(* Logix 5000 project; controller Sucrose_Main Emulate 5570 rev 20.12; software revision 20.01; part 11 of 30 *)
(* tags used below, declared in another part *)
   AI_E21_1 : REAL[8];   // Analog Input EN2T_FLX 192.168.1.21
   AI_E21_2 : REAL[8];   // Analog Input EN2T_FLX 192.168.1.21
   AI_E23_1 : REAL[8];   // Analog Input EN2T_FLX 192.168.1.23
   Alarm_ACK_Master_Timer : TIMER;
   ClearFault_Master : BOOL;
   DI_E20_2 : ALIAS FOR FLX_E20:2:I;   // Discrete Input EN2T_FLX 192.168.1.20
   DO_E24_3 : ALIAS FOR FLX_E24:3:O;   // Discrete Output EN2T_FLX 192.168.1.24
   FV230303_AOI : QSI_Flow_Valve;   // FV-23-03-03 SUCROSE TANK #3 OUTLET VALVE
   HEADER_FLOW_SP : DINT;
   ONESHOTBITS : INT[10];
   P230401_AOI : PF525_VFD_E_ENET;   // P-23-04-01 SUCROSE TRANSFER PUMP 1
   P230402_AOI : PF525_VFD_E_ENET;   // P-23-04-02 SUCROSE TRANSFER PUMP 2
   READ_FROM_SUCROSE_CIP : DINT[10];
   Rung_Comment : BOOL;
   Sucrose_MM_Enable : BOOL;
   SucroseCIP_FILTRATION_REMOTE : CIP_REMOTE;
   SucroseCIP_P230401_REMOTE : CIP_REMOTE;
   SucroseCIP_P230402_REMOTE : CIP_REMOTE;
   SucroseCIP_TK230301_REMOTE : CIP_REMOTE;
   SucroseDischarge : Area_Program;
   SucroseFiltration : Area_Program;
   SucroseTanks : Area_Program;
   temp_toggle : BOOL;
   toggle : BOOL;
(* DischargeArea_EN2T_IO_Discrete_DO_E24_3, continued *)

ROUTINE _11_FV230303   (* ladder *)
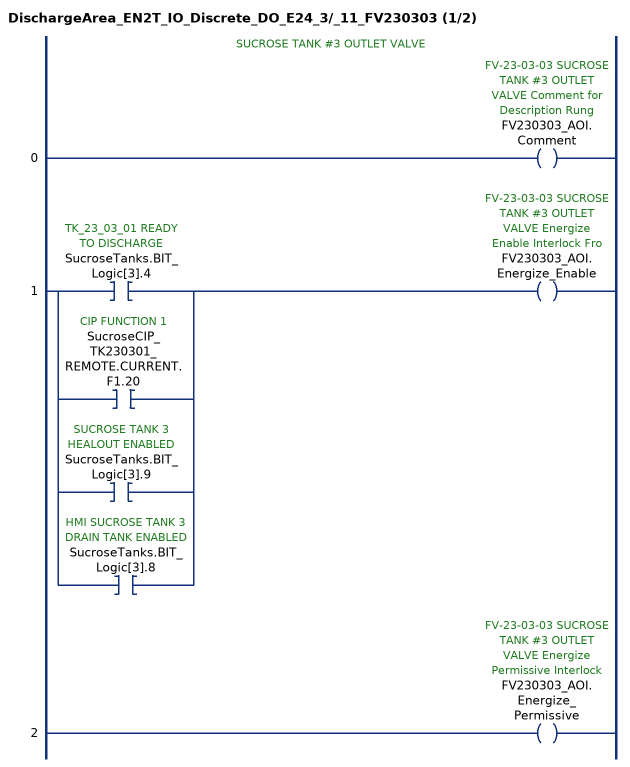
   // SUCROSE TANK #3 OUTLET VALVE
   0: OTE(FV230303_AOI.Comment);
   1: [XIC(SucroseTanks.BIT_Logic[3].4) ,XIC(SucroseCIP_TK230301_REMOTE.CURRENT.F1.20) ,XIC(SucroseTanks.BIT_Logic[3].9) ,XIC(SucroseTanks.BIT_Logic[3].8) ]OTE(FV230303_AOI.Energize_Enable);
   2: OTE(FV230303_AOI.Energize_Permissive);
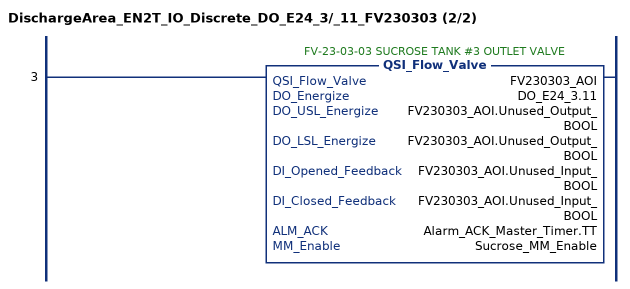
   3: QSI_Flow_Valve(FV230303_AOI,DO_E24_3.11,FV230303_AOI.Unused_Output_BOOL,FV230303_AOI.Unused_Output_BOOL,FV230303_AOI.Unused_Input_BOOL,FV230303_AOI.Unused_Input_BOOL,Alarm_ACK_Master_Timer.TT,Sucrose_MM_Enable);
END_ROUTINE

ROUTINE MainRoutine   (* ladder *)
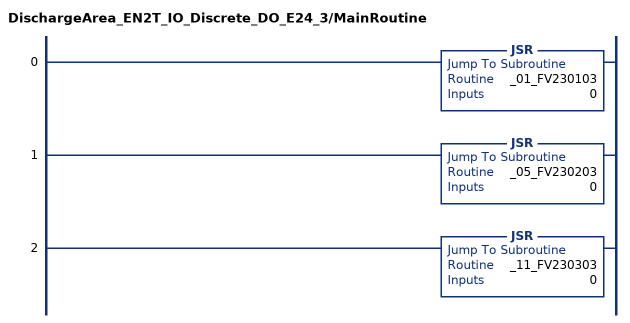
   0: JSR(_01_FV230103,0);
   1: JSR(_05_FV230203,0);
   2: JSR(_11_FV230303,0);
END_ROUTINE
END_PROGRAM

PROGRAM DischargeArea_EN2T_IO_Drives   (* main routine MainRoutine *)

ROUTINE E30_P230401   (* ladder *)
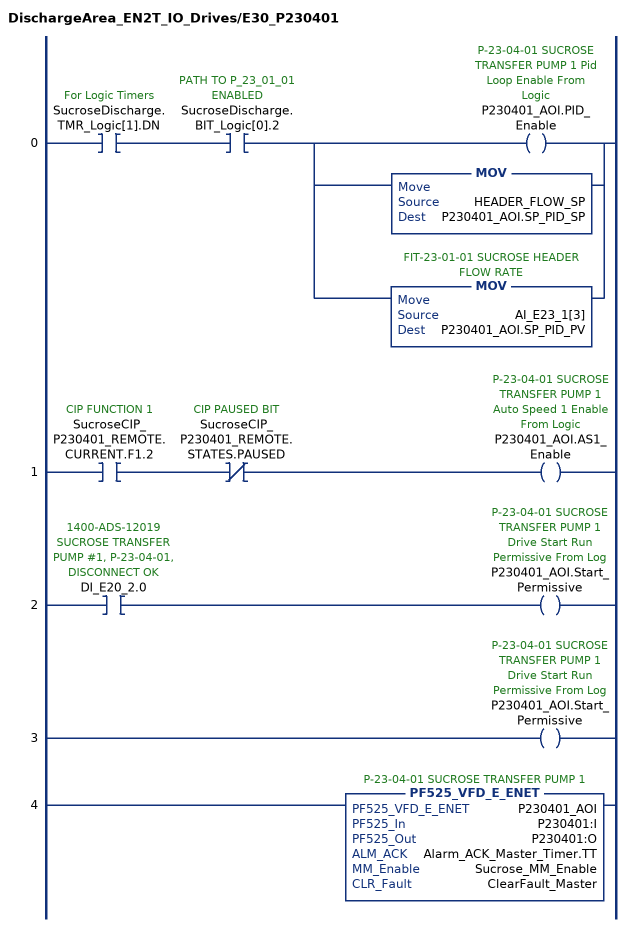
   0: XIC(SucroseDischarge.TMR_Logic[1].DN)XIC(SucroseDischarge.BIT_Logic[0].2)[OTE(P230401_AOI.PID_Enable) ,MOV(HEADER_FLOW_SP,P230401_AOI.SP_PID_SP) ,MOV(AI_E23_1[3],P230401_AOI.SP_PID_PV) ];
   1: XIC(SucroseCIP_P230401_REMOTE.CURRENT.F1.2)XIO(SucroseCIP_P230401_REMOTE.STATES.PAUSED)OTE(P230401_AOI.AS1_Enable);
   2: XIC(DI_E20_2.0)OTE(P230401_AOI.Start_Permissive);
   3: OTE(P230401_AOI.Start_Permissive);
   4: PF525_VFD_E_ENET(P230401_AOI,P230401:I,P230401:O,Alarm_ACK_Master_Timer.TT,Sucrose_MM_Enable,ClearFault_Master);
END_ROUTINE

ROUTINE E31_P200402   (* ladder *)
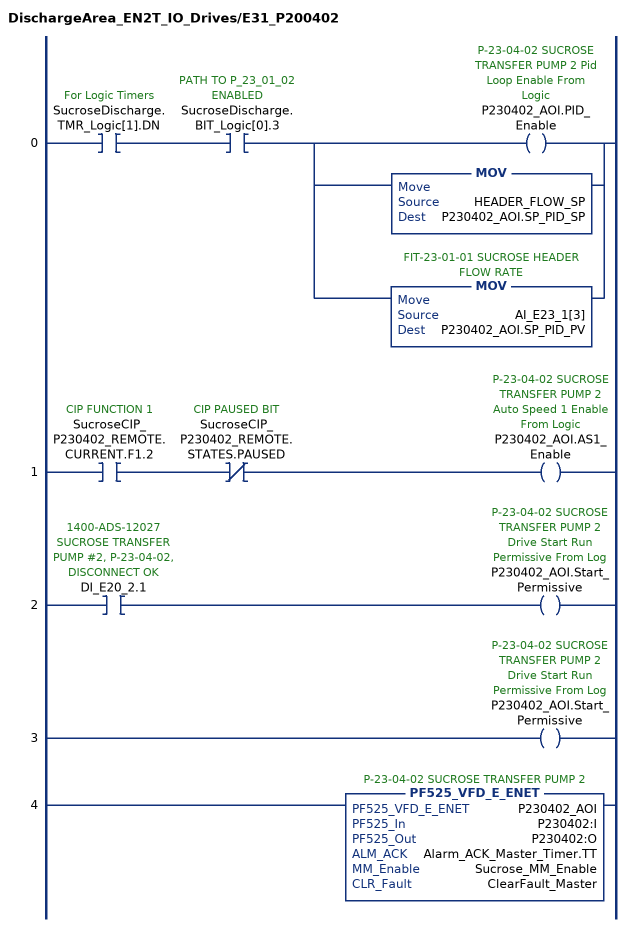
   0: XIC(SucroseDischarge.TMR_Logic[1].DN)XIC(SucroseDischarge.BIT_Logic[0].3)[OTE(P230402_AOI.PID_Enable) ,MOV(HEADER_FLOW_SP,P230402_AOI.SP_PID_SP) ,MOV(AI_E23_1[3],P230402_AOI.SP_PID_PV) ];
   1: XIC(SucroseCIP_P230402_REMOTE.CURRENT.F1.2)XIO(SucroseCIP_P230402_REMOTE.STATES.PAUSED)OTE(P230402_AOI.AS1_Enable);
   2: XIC(DI_E20_2.1)OTE(P230402_AOI.Start_Permissive);
   3: OTE(P230402_AOI.Start_Permissive);
   4: PF525_VFD_E_ENET(P230402_AOI,P230402:I,P230402:O,Alarm_ACK_Master_Timer.TT,Sucrose_MM_Enable,ClearFault_Master);
END_ROUTINE

ROUTINE MainRoutine   (* ladder *)
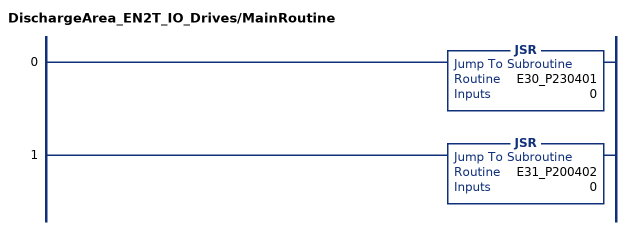
   0: JSR(E30_P230401,0);
   1: JSR(E31_P200402,0);
END_ROUTINE
END_PROGRAM

PROGRAM FiltrationArea_AutoLogic   (* main routine MainRoutine *)

ROUTINE Alarm_Logic   (* ladder *)
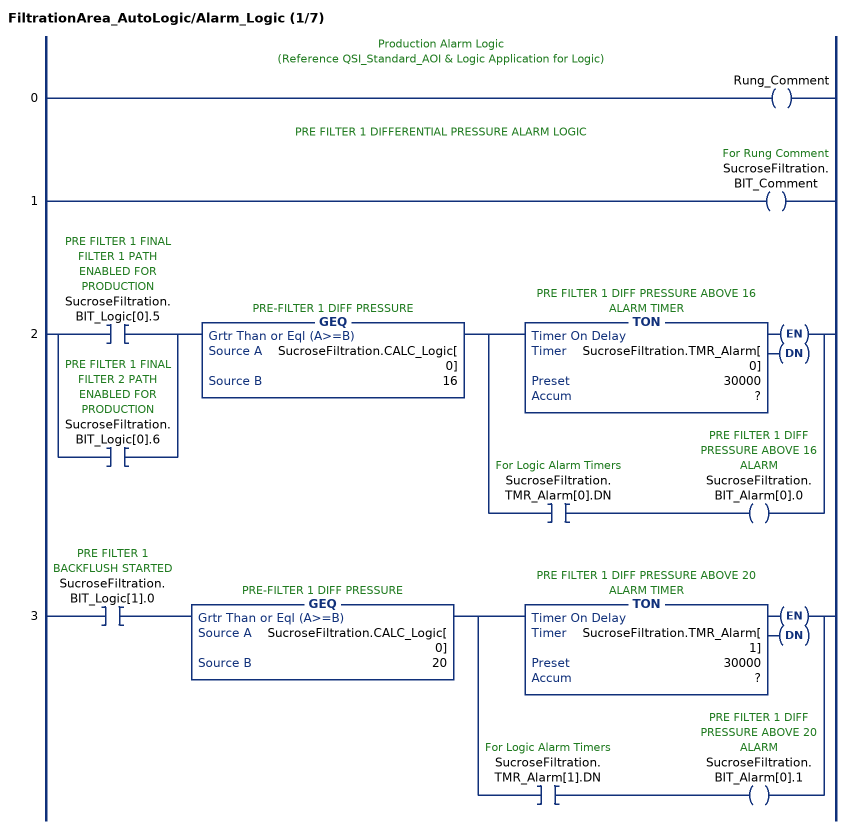
   // Production Alarm Logic
   // (Reference QSI_Standard_AOI & Logic Application for Logic)
   0: OTE(Rung_Comment);
   // PRE FILTER 1 DIFFERENTIAL PRESSURE ALARM LOGIC
   1: OTE(SucroseFiltration.BIT_Comment);
   2: [XIC(SucroseFiltration.BIT_Logic[0].5) ,XIC(SucroseFiltration.BIT_Logic[0].6) ]GEQ(SucroseFiltration.CALC_Logic[0],16)[TON(SucroseFiltration.TMR_Alarm[0],?,?) ,XIC(SucroseFiltration.TMR_Alarm[0].DN) OTE(SucroseFiltration.BIT_Alarm[0].0) ];
   3: XIC(SucroseFiltration.BIT_Logic[1].0)GEQ(SucroseFiltration.CALC_Logic[0],20)[TON(SucroseFiltration.TMR_Alarm[1],?,?) ,XIC(SucroseFiltration.TMR_Alarm[1].DN) OTE(SucroseFiltration.BIT_Alarm[0].1) ];
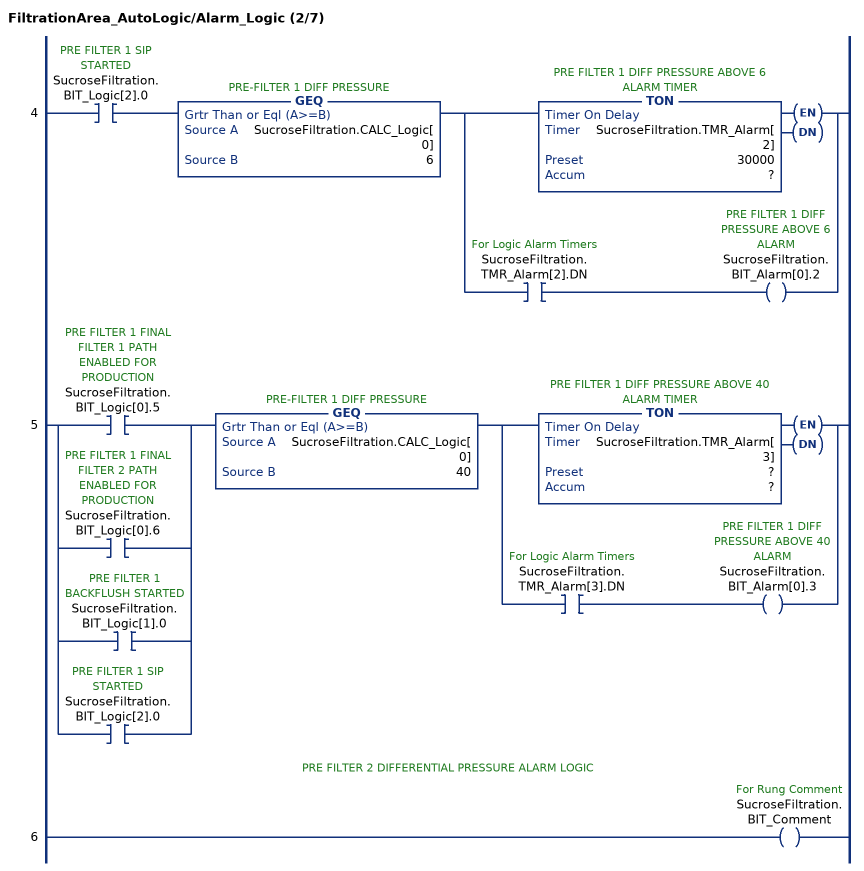
   4: XIC(SucroseFiltration.BIT_Logic[2].0)GEQ(SucroseFiltration.CALC_Logic[0],6)[TON(SucroseFiltration.TMR_Alarm[2],?,?) ,XIC(SucroseFiltration.TMR_Alarm[2].DN) OTE(SucroseFiltration.BIT_Alarm[0].2) ];
   5: [XIC(SucroseFiltration.BIT_Logic[0].5) ,XIC(SucroseFiltration.BIT_Logic[0].6) ,XIC(SucroseFiltration.BIT_Logic[1].0) ,XIC(SucroseFiltration.BIT_Logic[2].0) ]GEQ(SucroseFiltration.CALC_Logic[0],40)[TON(SucroseFiltration.TMR_Alarm[3],?,?) ,XIC(SucroseFiltration.TMR_Alarm[3].DN) OTE(SucroseFiltration.BIT_Alarm[0].3) ];
   // PRE FILTER 2 DIFFERENTIAL PRESSURE ALARM LOGIC
   6: OTE(SucroseFiltration.BIT_Comment);
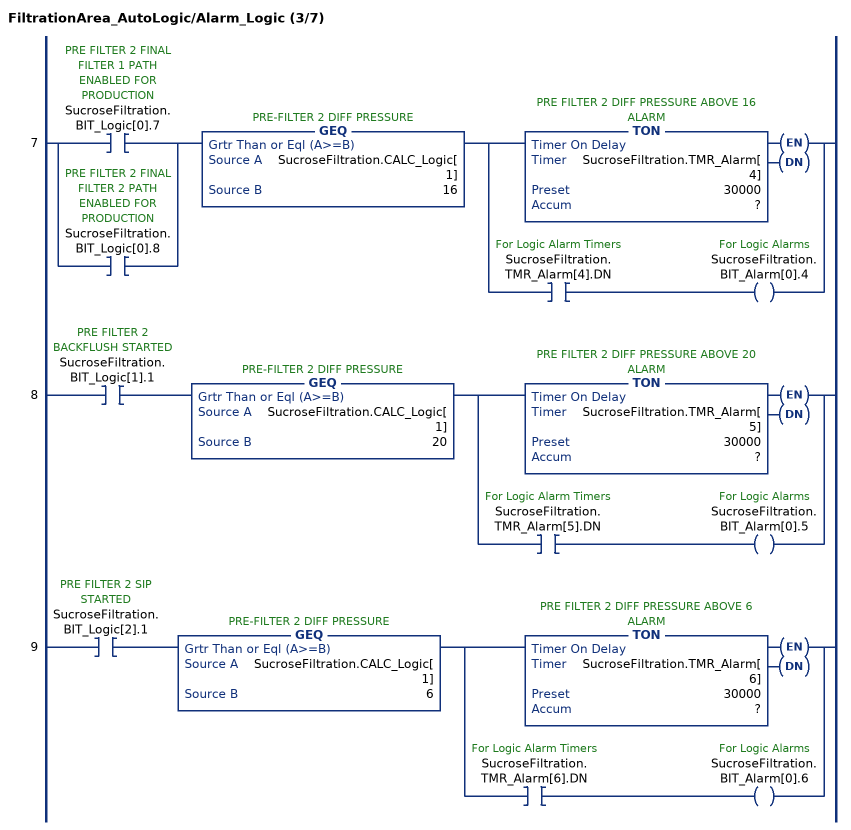
   7: [XIC(SucroseFiltration.BIT_Logic[0].7) ,XIC(SucroseFiltration.BIT_Logic[0].8) ]GEQ(SucroseFiltration.CALC_Logic[1],16)[TON(SucroseFiltration.TMR_Alarm[4],?,?) ,XIC(SucroseFiltration.TMR_Alarm[4].DN) OTE(SucroseFiltration.BIT_Alarm[0].4) ];
   8: XIC(SucroseFiltration.BIT_Logic[1].1)GEQ(SucroseFiltration.CALC_Logic[1],20)[TON(SucroseFiltration.TMR_Alarm[5],?,?) ,XIC(SucroseFiltration.TMR_Alarm[5].DN) OTE(SucroseFiltration.BIT_Alarm[0].5) ];
   9: XIC(SucroseFiltration.BIT_Logic[2].1)GEQ(SucroseFiltration.CALC_Logic[1],6)[TON(SucroseFiltration.TMR_Alarm[6],?,?) ,XIC(SucroseFiltration.TMR_Alarm[6].DN) OTE(SucroseFiltration.BIT_Alarm[0].6) ];
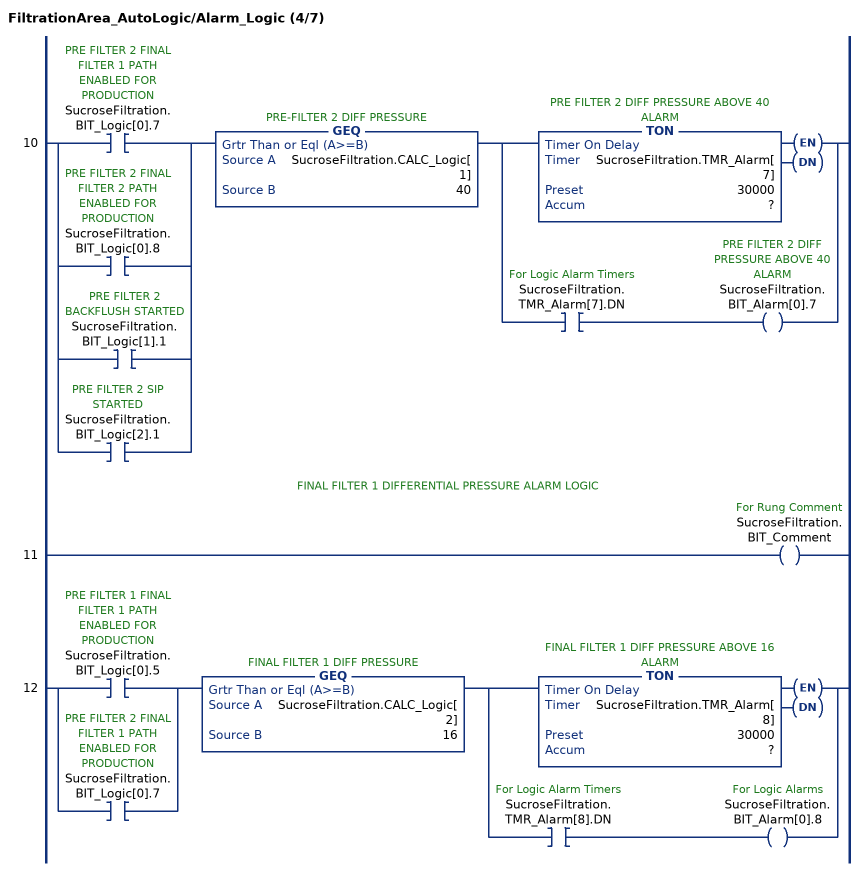
   10: [XIC(SucroseFiltration.BIT_Logic[0].7) ,XIC(SucroseFiltration.BIT_Logic[0].8) ,XIC(SucroseFiltration.BIT_Logic[1].1) ,XIC(SucroseFiltration.BIT_Logic[2].1) ]GEQ(SucroseFiltration.CALC_Logic[1],40)[TON(SucroseFiltration.TMR_Alarm[7],?,?) ,XIC(SucroseFiltration.TMR_Alarm[7].DN) OTE(SucroseFiltration.BIT_Alarm[0].7) ];
   // FINAL FILTER 1 DIFFERENTIAL PRESSURE ALARM LOGIC
   11: OTE(SucroseFiltration.BIT_Comment);
   12: [XIC(SucroseFiltration.BIT_Logic[0].5) ,XIC(SucroseFiltration.BIT_Logic[0].7) ]GEQ(SucroseFiltration.CALC_Logic[2],16)[TON(SucroseFiltration.TMR_Alarm[8],?,?) ,XIC(SucroseFiltration.TMR_Alarm[8].DN) OTE(SucroseFiltration.BIT_Alarm[0].8) ];
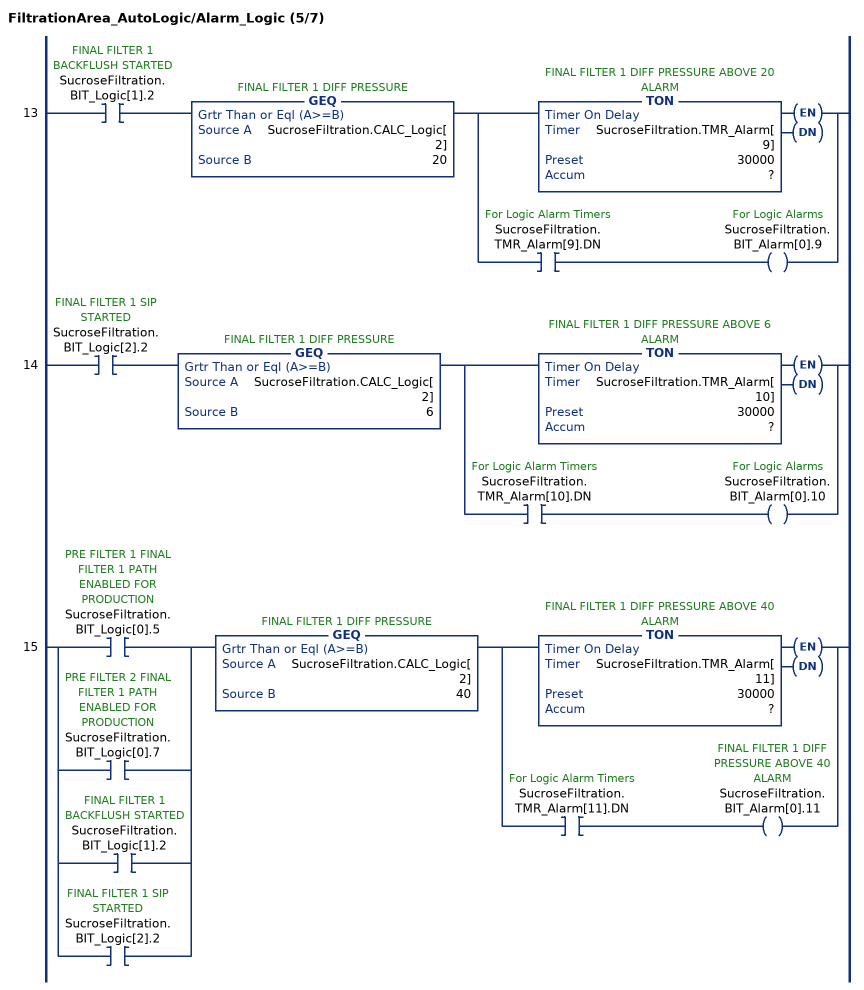
   13: XIC(SucroseFiltration.BIT_Logic[1].2)GEQ(SucroseFiltration.CALC_Logic[2],20)[TON(SucroseFiltration.TMR_Alarm[9],?,?) ,XIC(SucroseFiltration.TMR_Alarm[9].DN) OTE(SucroseFiltration.BIT_Alarm[0].9) ];
   14: XIC(SucroseFiltration.BIT_Logic[2].2)GEQ(SucroseFiltration.CALC_Logic[2],6)[TON(SucroseFiltration.TMR_Alarm[10],?,?) ,XIC(SucroseFiltration.TMR_Alarm[10].DN) OTE(SucroseFiltration.BIT_Alarm[0].10) ];
   15: [XIC(SucroseFiltration.BIT_Logic[0].5) ,XIC(SucroseFiltration.BIT_Logic[0].7) ,XIC(SucroseFiltration.BIT_Logic[1].2) ,XIC(SucroseFiltration.BIT_Logic[2].2) ]GEQ(SucroseFiltration.CALC_Logic[2],40)[TON(SucroseFiltration.TMR_Alarm[11],?,?) ,XIC(SucroseFiltration.TMR_Alarm[11].DN) OTE(SucroseFiltration.BIT_Alarm[0].11) ];
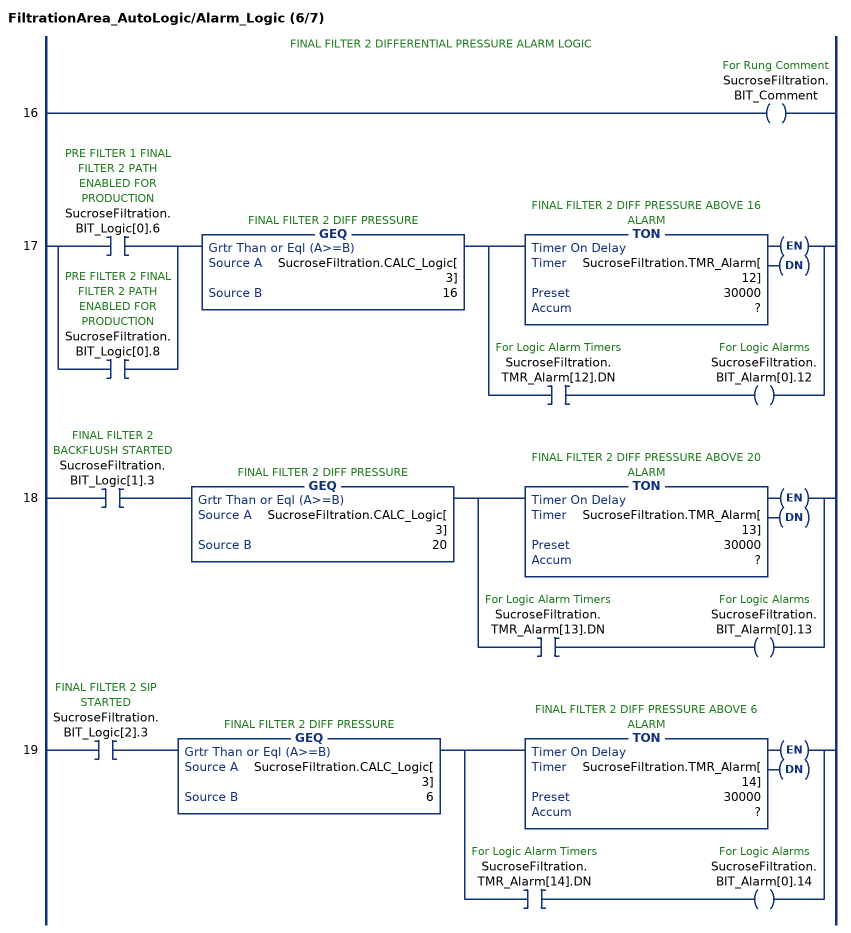
   // FINAL FILTER 2 DIFFERENTIAL PRESSURE ALARM LOGIC
   16: OTE(SucroseFiltration.BIT_Comment);
   17: [XIC(SucroseFiltration.BIT_Logic[0].6) ,XIC(SucroseFiltration.BIT_Logic[0].8) ]GEQ(SucroseFiltration.CALC_Logic[3],16)[TON(SucroseFiltration.TMR_Alarm[12],?,?) ,XIC(SucroseFiltration.TMR_Alarm[12].DN) OTE(SucroseFiltration.BIT_Alarm[0].12) ];
   18: XIC(SucroseFiltration.BIT_Logic[1].3)GEQ(SucroseFiltration.CALC_Logic[3],20)[TON(SucroseFiltration.TMR_Alarm[13],?,?) ,XIC(SucroseFiltration.TMR_Alarm[13].DN) OTE(SucroseFiltration.BIT_Alarm[0].13) ];
   19: XIC(SucroseFiltration.BIT_Logic[2].3)GEQ(SucroseFiltration.CALC_Logic[3],6)[TON(SucroseFiltration.TMR_Alarm[14],?,?) ,XIC(SucroseFiltration.TMR_Alarm[14].DN) OTE(SucroseFiltration.BIT_Alarm[0].14) ];
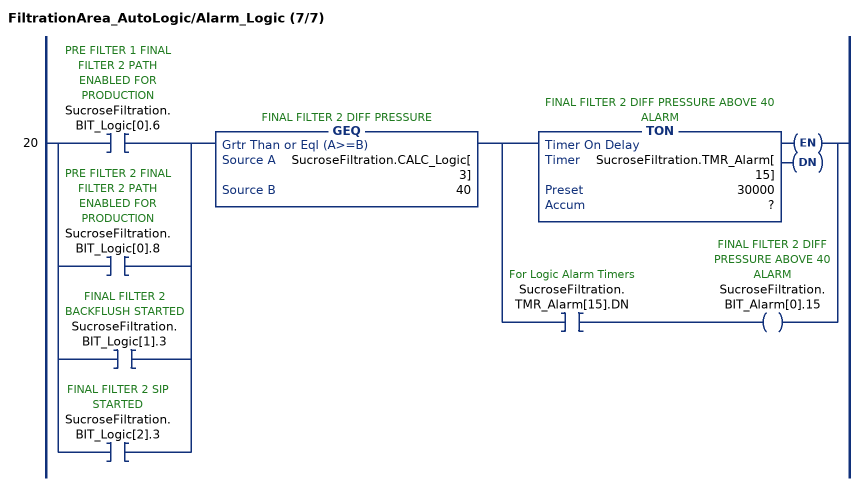
   20: [XIC(SucroseFiltration.BIT_Logic[0].6) ,XIC(SucroseFiltration.BIT_Logic[0].8) ,XIC(SucroseFiltration.BIT_Logic[1].3) ,XIC(SucroseFiltration.BIT_Logic[2].3) ]GEQ(SucroseFiltration.CALC_Logic[3],40)[TON(SucroseFiltration.TMR_Alarm[15],?,?) ,XIC(SucroseFiltration.TMR_Alarm[15].DN) OTE(SucroseFiltration.BIT_Alarm[0].15) ];
END_ROUTINE

ROUTINE Control_Logic   (* ladder *)
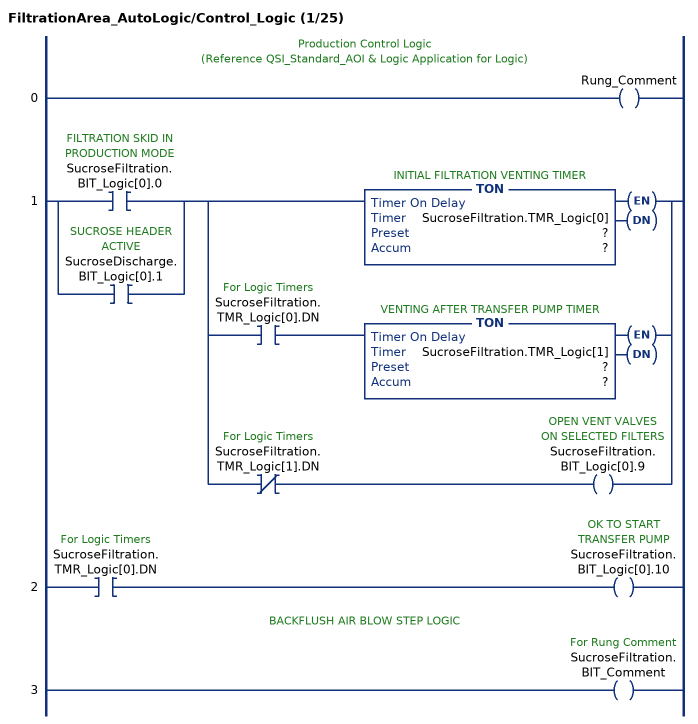
   // Production Control Logic
   // (Reference QSI_Standard_AOI & Logic Application for Logic)
   0: OTE(Rung_Comment);
   1: [XIC(SucroseFiltration.BIT_Logic[0].0) ,XIC(SucroseDischarge.BIT_Logic[0].1) ][TON(SucroseFiltration.TMR_Logic[0],?,?) ,XIC(SucroseFiltration.TMR_Logic[0].DN) TON(SucroseFiltration.TMR_Logic[1],?,?) ,XIO(SucroseFiltration.TMR_Logic[1].DN) OTE(SucroseFiltration.BIT_Logic[0].9) ];
   2: XIC(SucroseFiltration.TMR_Logic[0].DN)OTE(SucroseFiltration.BIT_Logic[0].10);
   // BACKFLUSH AIR BLOW STEP LOGIC
   3: OTE(SucroseFiltration.BIT_Comment);
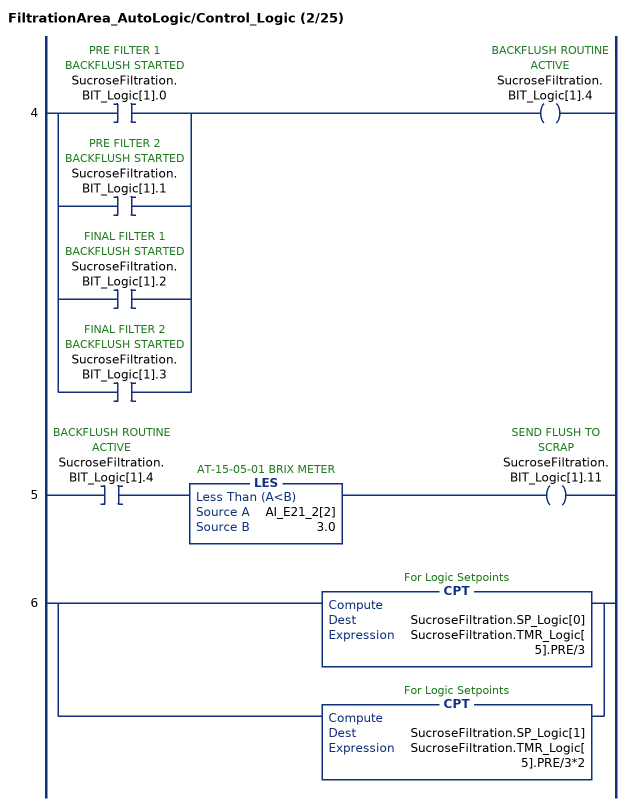
   4: [XIC(SucroseFiltration.BIT_Logic[1].0) ,XIC(SucroseFiltration.BIT_Logic[1].1) ,XIC(SucroseFiltration.BIT_Logic[1].2) ,XIC(SucroseFiltration.BIT_Logic[1].3) ]OTE(SucroseFiltration.BIT_Logic[1].4);
   5: XIC(SucroseFiltration.BIT_Logic[1].4)LES(AI_E21_2[2],3.0)OTE(SucroseFiltration.BIT_Logic[1].11);
   6: [CPT(SucroseFiltration.SP_Logic[0],SucroseFiltration.TMR_Logic[5].PRE/3) ,CPT(SucroseFiltration.SP_Logic[1],SucroseFiltration.TMR_Logic[5].PRE/3*2) ];
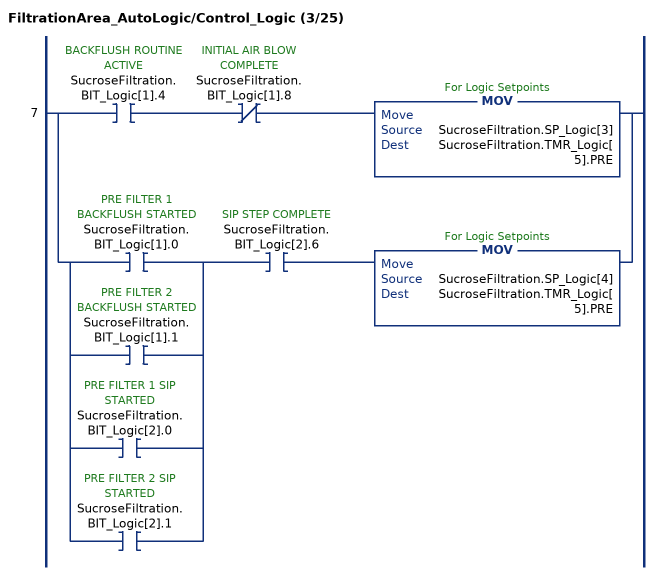
   7: [XIC(SucroseFiltration.BIT_Logic[1].4) XIO(SucroseFiltration.BIT_Logic[1].8) MOV(SucroseFiltration.SP_Logic[3],SucroseFiltration.TMR_Logic[5].PRE) ,[XIC(SucroseFiltration.BIT_Logic[1].0) ,XIC(SucroseFiltration.BIT_Logic[1].1) ,XIC(SucroseFiltration.BIT_Logic[2].0) ,XIC(SucroseFiltration.BIT_Logic[2].1) ] XIC(SucroseFiltration.BIT_Logic[2].6) MOV(SucroseFiltration.SP_Logic[4],SucroseFiltration.TMR_Logic[5].PRE) ];
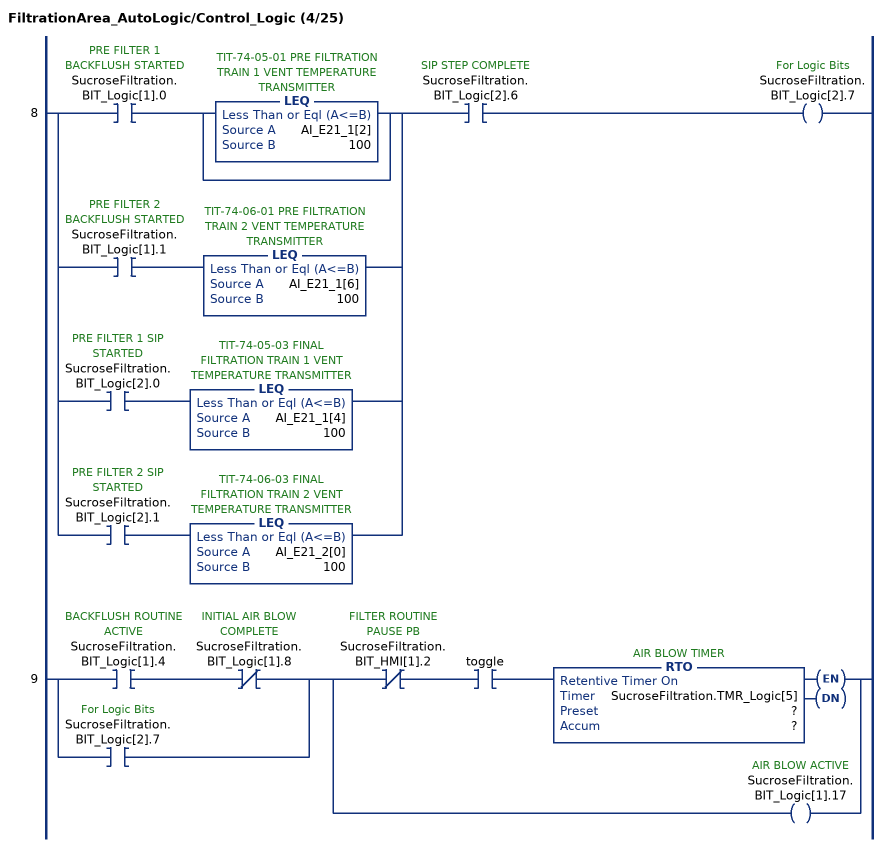
   8: [XIC(SucroseFiltration.BIT_Logic[1].0) [LEQ(AI_E21_1[2],100) ,] ,XIC(SucroseFiltration.BIT_Logic[1].1) LEQ(AI_E21_1[6],100) ,XIC(SucroseFiltration.BIT_Logic[2].0) LEQ(AI_E21_1[4],100) ,XIC(SucroseFiltration.BIT_Logic[2].1) LEQ(AI_E21_2[0],100) ]XIC(SucroseFiltration.BIT_Logic[2].6)OTE(SucroseFiltration.BIT_Logic[2].7);
   9: [XIC(SucroseFiltration.BIT_Logic[1].4) XIO(SucroseFiltration.BIT_Logic[1].8) ,XIC(SucroseFiltration.BIT_Logic[2].7) ][XIO(SucroseFiltration.BIT_HMI[1].2) XIC(toggle) RTO(SucroseFiltration.TMR_Logic[5],?,?) ,OTE(SucroseFiltration.BIT_Logic[1].17) ];
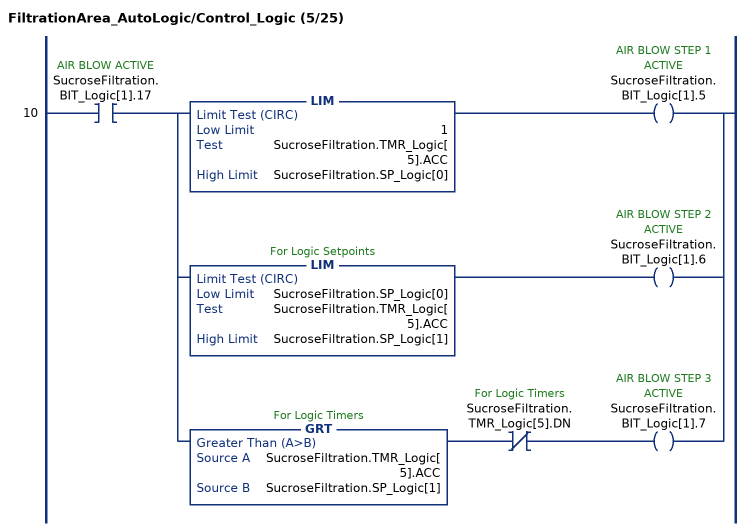
   10: XIC(SucroseFiltration.BIT_Logic[1].17)[LIM(1,SucroseFiltration.TMR_Logic[5].ACC,SucroseFiltration.SP_Logic[0]) OTE(SucroseFiltration.BIT_Logic[1].5) ,LIM(SucroseFiltration.SP_Logic[0],SucroseFiltration.TMR_Logic[5].ACC,SucroseFiltration.SP_Logic[1]) OTE(SucroseFiltration.BIT_Logic[1].6) ,GRT(SucroseFiltration.TMR_Logic[5].ACC,SucroseFiltration.SP_Logic[1]) XIO(SucroseFiltration.TMR_Logic[5].DN) OTE(SucroseFiltration.BIT_Logic[1].7) ];
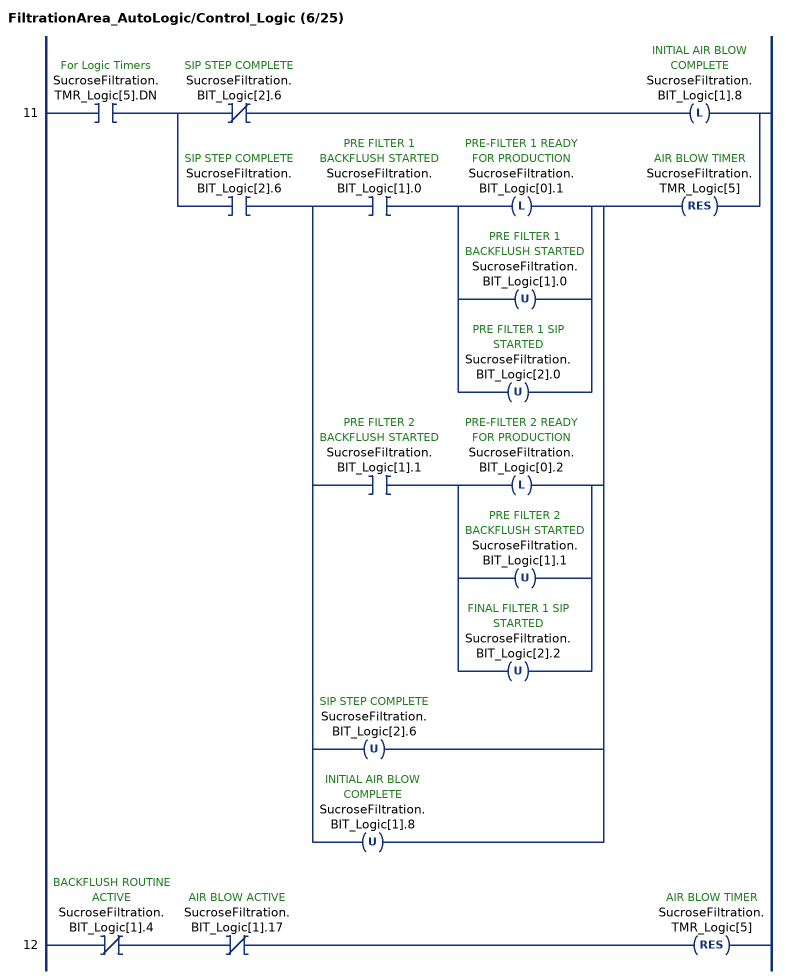
   11: XIC(SucroseFiltration.TMR_Logic[5].DN)[XIO(SucroseFiltration.BIT_Logic[2].6) OTL(SucroseFiltration.BIT_Logic[1].8) ,XIC(SucroseFiltration.BIT_Logic[2].6) [XIC(SucroseFiltration.BIT_Logic[1].0) [OTL(SucroseFiltration.BIT_Logic[0].1) ,OTU(SucroseFiltration.BIT_Logic[1].0) ,OTU(SucroseFiltration.BIT_Logic[2].0) ] ,XIC(SucroseFiltration.BIT_Logic[1].1) [OTL(SucroseFiltration.BIT_Logic[0].2) ,OTU(SucroseFiltration.BIT_Logic[1].1) ,OTU(SucroseFiltration.BIT_Logic[2].2) ] ,OTU(SucroseFiltration.BIT_Logic[2].6) ,OTU(SucroseFiltration.BIT_Logic[1].8) ] RES(SucroseFiltration.TMR_Logic[5]) ];
   12: XIO(SucroseFiltration.BIT_Logic[1].4)XIO(SucroseFiltration.BIT_Logic[1].17)RES(SucroseFiltration.TMR_Logic[5]);
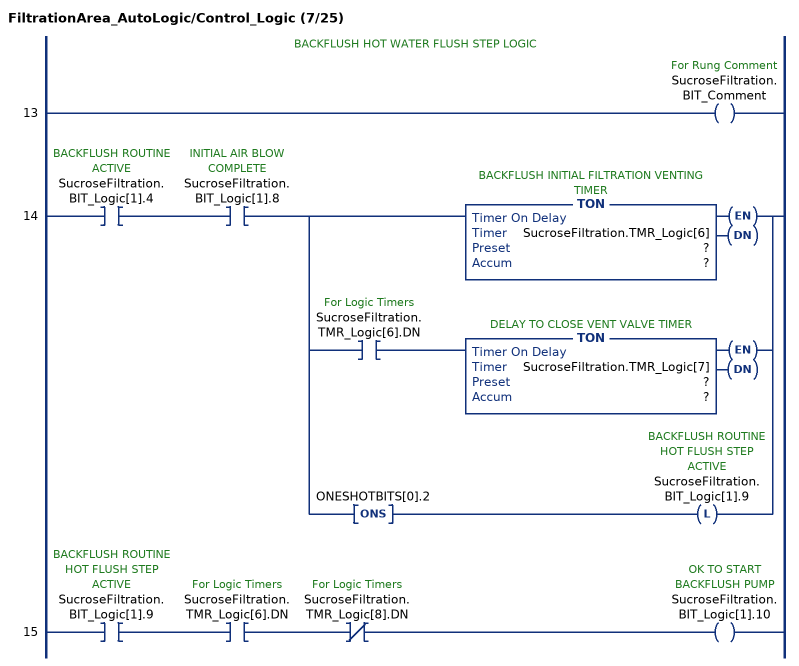
   // BACKFLUSH HOT WATER FLUSH STEP LOGIC
   13: OTE(SucroseFiltration.BIT_Comment);
   14: XIC(SucroseFiltration.BIT_Logic[1].4)XIC(SucroseFiltration.BIT_Logic[1].8)[TON(SucroseFiltration.TMR_Logic[6],?,?) ,XIC(SucroseFiltration.TMR_Logic[6].DN) TON(SucroseFiltration.TMR_Logic[7],?,?) ,ONS(ONESHOTBITS[0].2) OTL(SucroseFiltration.BIT_Logic[1].9) ];
   15: XIC(SucroseFiltration.BIT_Logic[1].9)XIC(SucroseFiltration.TMR_Logic[6].DN)XIO(SucroseFiltration.TMR_Logic[8].DN)OTE(SucroseFiltration.BIT_Logic[1].10);
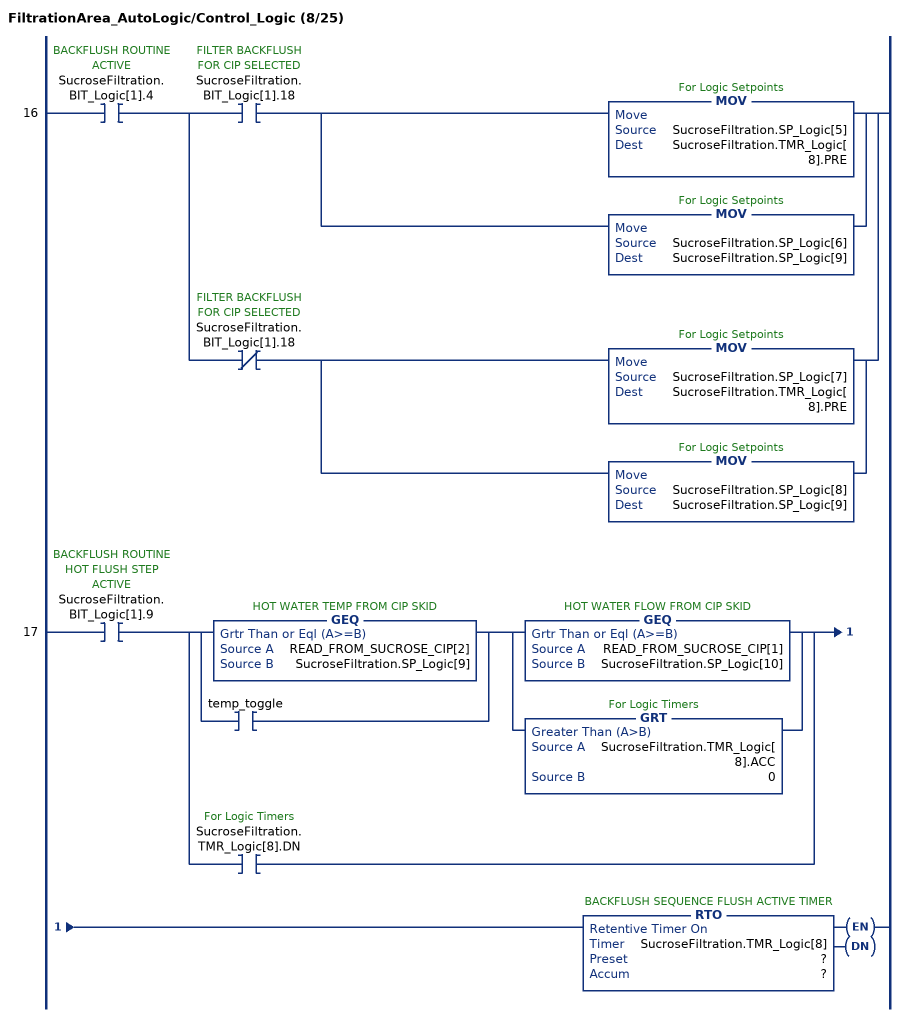
   16: XIC(SucroseFiltration.BIT_Logic[1].4)[XIC(SucroseFiltration.BIT_Logic[1].18) [MOV(SucroseFiltration.SP_Logic[5],SucroseFiltration.TMR_Logic[8].PRE) ,MOV(SucroseFiltration.SP_Logic[6],SucroseFiltration.SP_Logic[9]) ] ,XIO(SucroseFiltration.BIT_Logic[1].18) [MOV(SucroseFiltration.SP_Logic[7],SucroseFiltration.TMR_Logic[8].PRE) ,MOV(SucroseFiltration.SP_Logic[8],SucroseFiltration.SP_Logic[9]) ] ];
   17: XIC(SucroseFiltration.BIT_Logic[1].9)[[GEQ(READ_FROM_SUCROSE_CIP[2],SucroseFiltration.SP_Logic[9]) ,XIC(temp_toggle) ] [GEQ(READ_FROM_SUCROSE_CIP[1],SucroseFiltration.SP_Logic[10]) ,GRT(SucroseFiltration.TMR_Logic[8].ACC,0) ] ,XIC(SucroseFiltration.TMR_Logic[8].DN) ]RTO(SucroseFiltration.TMR_Logic[8],?,?);
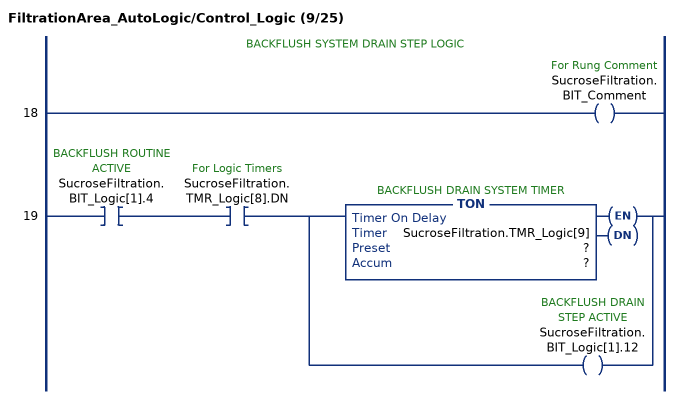
   // BACKFLUSH SYSTEM DRAIN STEP LOGIC
   18: OTE(SucroseFiltration.BIT_Comment);
   19: XIC(SucroseFiltration.BIT_Logic[1].4)XIC(SucroseFiltration.TMR_Logic[8].DN)[TON(SucroseFiltration.TMR_Logic[9],?,?) ,OTE(SucroseFiltration.BIT_Logic[1].12) ];
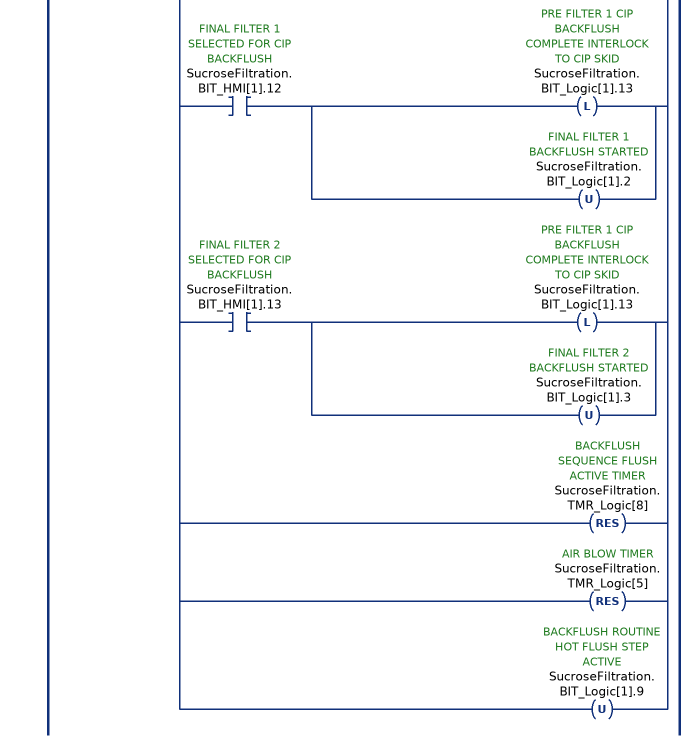
   20: XIC(SucroseFiltration.TMR_Logic[9].DN)[XIC(SucroseFiltration.BIT_Logic[1].0) CTU(SucroseFiltration.CTR_Logic[0],?,?) ,XIC(SucroseFiltration.BIT_Logic[1].1) CTU(SucroseFiltration.CTR_Logic[1],?,?) ,XIC(SucroseFiltration.BIT_Logic[1].2) CTU(SucroseFiltration.CTR_Logic[2],?,?) ,XIC(SucroseFiltration.BIT_Logic[1].3) CTU(SucroseFiltration.CTR_Logic[3],?,?) ,XIC(SucroseFiltration.BIT_HMI[1].10) [OTL(SucroseFiltration.BIT_Logic[1].13) ,OTU(SucroseFiltration.BIT_Logic[1].0) ] ,XIC(SucroseFiltration.BIT_HMI[1].11) [OTL(SucroseFiltration.BIT_Logic[1].13) ,OTU(SucroseFiltration.BIT_Logic[1].1) ] ,XIC(SucroseFiltration.BIT_HMI[1].12) [OTL(SucroseFiltration.BIT_Logic[1].13) ,OTU(SucroseFiltration.BIT_Logic[1].2) ] ,XIC(SucroseFiltration.BIT_HMI[1].13) [OTL(SucroseFiltration.BIT_Logic[1].13) ,OTU(SucroseFiltration.BIT_Logic[1].3) ] ,RES(SucroseFiltration.TMR_Logic[8]) ,RES(SucroseFiltration.TMR_Logic[5]) ,OTU(SucroseFiltration.BIT_Logic[1].9) ];
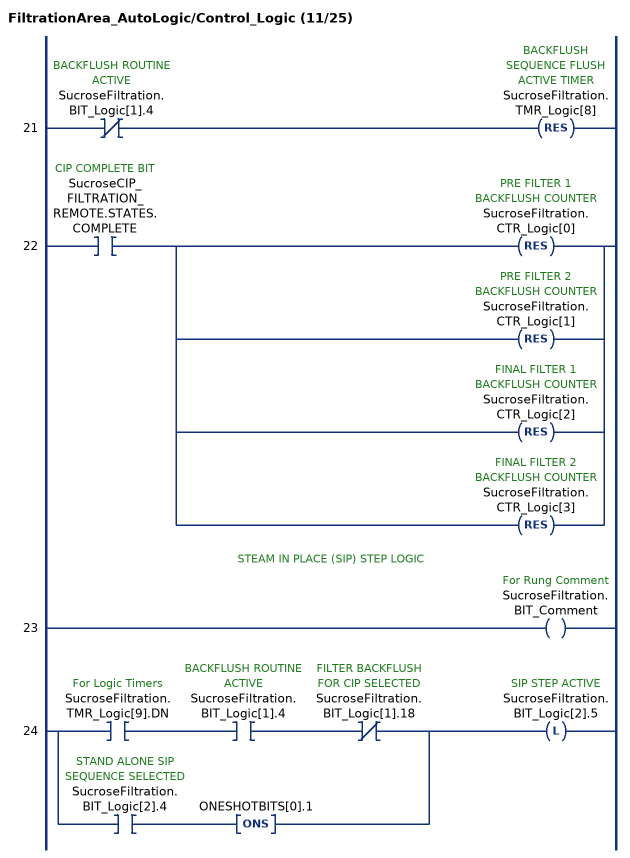
   21: XIO(SucroseFiltration.BIT_Logic[1].4)RES(SucroseFiltration.TMR_Logic[8]);
   22: XIC(SucroseCIP_FILTRATION_REMOTE.STATES.COMPLETE)[RES(SucroseFiltration.CTR_Logic[0]) ,RES(SucroseFiltration.CTR_Logic[1]) ,RES(SucroseFiltration.CTR_Logic[2]) ,RES(SucroseFiltration.CTR_Logic[3]) ];
   // STEAM IN PLACE (SIP) STEP LOGIC
   23: OTE(SucroseFiltration.BIT_Comment);
   24: [XIC(SucroseFiltration.TMR_Logic[9].DN) XIC(SucroseFiltration.BIT_Logic[1].4) XIO(SucroseFiltration.BIT_Logic[1].18) ,XIC(SucroseFiltration.BIT_Logic[2].4) ONS(ONESHOTBITS[0].1) ]OTL(SucroseFiltration.BIT_Logic[2].5);
